// TIA Portal V19 export
DATA_BLOCK "PrjConfig_A04"   // DB212
// stored: MemoryReserve 100
   VAR
      Area04_Main : "AreaConfig";
   END_VAR
   VAR RETAIN
      A0303 : Struct
         Spalla : Struct
            Testa : Struct
               Ax : "Positioning_DOL_Machine_Config";
               DelayMissingCondition { ExternalAccessible := 'False'; ExternalVisible := 'False'; ExternalWritable := 'False'} : Time := T#0MS;
            END_STRUCT;
            Coda : Struct
               Ax : "Positioning_DOL_Machine_Config";
               DelayMissingCondition { ExternalAccessible := 'False'; ExternalVisible := 'False'; ExternalWritable := 'False'} : Time := T#0MS;
            END_STRUCT;
         END_STRUCT;
         Spintore : Struct
            Testa : Struct
               Vrt : "ValveMachine_Config";
               Orz { S7_SetPoint := 'True'} : "ValveMachine_Config";
            END_STRUCT;
            Coda : Struct
               Vrt : "ValveMachine_Config";
               Orz { S7_SetPoint := 'True'} : "ValveMachine_Config";
            END_STRUCT;
            DelayMissingCondition { ExternalAccessible := 'False'; ExternalVisible := 'False'; ExternalWritable := 'False'} : Time := T#0MS;
         END_STRUCT;
         TraslazioneStrato : Struct
            Testa : Struct
               Ax { S7_SetPoint := 'True'} : "Positioning_EPOS_Machine_Config_NEW";
               Manip_Sostegno { S7_SetPoint := 'True'} : "ValveMachine_Config";
               Manip_Pareggiatore { S7_SetPoint := 'True'} : "ValveMachine_Config";
               SostegnoVrt { S7_SetPoint := 'True'} : "ValveMachine_Config";
            END_STRUCT;
            Coda : Struct
               Ax { S7_SetPoint := 'True'} : "Positioning_EPOS_Machine_Config_NEW";
               Manip_Sostegno { S7_SetPoint := 'True'} : "ValveMachine_Config";
               Manip_Pareggiatore { S7_SetPoint := 'True'} : "ValveMachine_Config";
               SostegnoVrt { S7_SetPoint := 'True'} : "ValveMachine_Config";
               DelayMissingCondition { ExternalAccessible := 'False'; ExternalVisible := 'False'; ExternalWritable := 'False'} : Time := T#0MS;
            END_STRUCT;
            DelayMissingCondition { ExternalAccessible := 'False'; ExternalVisible := 'False'; ExternalWritable := 'False'} : Time := T#2S;
         END_STRUCT;
         Sollevamento : Struct
            Testa : Struct
               Ax : "Positioning_DOL_Machine_Config";
            END_STRUCT;
            Coda : Struct
               Ax : "Positioning_DOL_Machine_Config";
            END_STRUCT;
            DelayMissingCondition { ExternalAccessible := 'False'; ExternalVisible := 'False'; ExternalWritable := 'False'} : Time := T#0MS;
         END_STRUCT;
         Sostegno : Struct
            Testa : Struct
               Ax : "Positioning_DOL_Machine_Config";
               V_1 { S7_SetPoint := 'True'} : "ValveMachine_Config";
               V_2 { S7_SetPoint := 'True'} : "ValveMachine_Config";
               DelayMissingCondition { ExternalAccessible := 'False'; ExternalVisible := 'False'; ExternalWritable := 'False'} : Time := T#0MS;
            END_STRUCT;
            Coda : Struct
               Ax : "Positioning_DOL_Machine_Config";
               V_1 { S7_SetPoint := 'True'} : "ValveMachine_Config";
               V_2 { S7_SetPoint := 'True'} : "ValveMachine_Config";
               DelayMissingCondition { ExternalAccessible := 'False'; ExternalVisible := 'False'; ExternalWritable := 'False'} : Time := T#0MS;
            END_STRUCT;
         END_STRUCT;
      END_STRUCT;
      A0304 : Struct
         Navetta : Struct
            Testa : Struct
               Ax : "Positioning_DOL_Machine_Config";
               PalettiEsterni { S7_SetPoint := 'True'} : "ValveMachine_Config";
               PalettiInterni { S7_SetPoint := 'True'} : "ValveMachine_Config";
            END_STRUCT;
            Coda : Struct
               Ax : "Positioning_DOL_Machine_Config";
               PalettiEsterni { S7_SetPoint := 'True'} : "ValveMachine_Config";
               PalettiInterni { S7_SetPoint := 'True'} : "ValveMachine_Config";
            END_STRUCT;
            DelayMissingCondition { ExternalAccessible := 'False'; ExternalVisible := 'False'; ExternalWritable := 'False'} : Time := T#0MS;
         END_STRUCT;
      END_STRUCT;
   END_VAR
BEGIN
   Area04_Main.TimeOutStopImmediate := T#1S_500MS;
   Area04_Main.TimeOutStopInPhase := T#10S;
   Area04_Main.TimeOutStopProgrammed := T#5M;
   Area04_Main.TimeOutResetAlarms := T#1S;
   A0303.Spalla.Testa.Ax.DelayMissingCondition := T#3S;
   A0303.Spalla.Testa.Ax.CyclicOBTime_ms := 10.0;
   A0303.Spalla.Testa.Ax.Ax.limitMinus := 83.0;
   A0303.Spalla.Testa.Ax.Ax.limitPlus := 2455.0;
   A0303.Spalla.Testa.Ax.Ax.Backlash := 0.0;
   A0303.Spalla.Testa.Ax.Ax.BacklashActivation := FALSE;
   A0303.Spalla.Testa.Ax.Ax.ToleranceWindow := 0.1;
   A0303.Spalla.Testa.Ax.Ax.ToleranceWindowDelay := T#100MS;
   A0303.Spalla.Testa.Ax.Ax.PreCutOff := 0.0;
   A0303.Spalla.Testa.Ax.Ax.PreEndLowSpeed := 0.0;
   A0303.Spalla.Testa.Ax.Ax.PreEndMedSpeed := 0.0;
   A0303.Spalla.Testa.Ax.Ax.ChangeDirectionDelay := T#0MS;
   A0303.Spalla.Testa.Ax.Ax.StandstillVelocity := 0.5;
   A0303.Spalla.Testa.Ax.Ax.StandStillDelay := T#100MS;
   A0303.Spalla.Testa.Ax.Ax.HomingDirection := FALSE;
   A0303.Spalla.Testa.Ax.Ax.RecallTime := 0.0;
   A0303.Spalla.Testa.Ax.Ax.VelocityFilter_T := 10.0;
   A0303.Spalla.Testa.Ax.Ax.VelocityMeasUnit := 2;
   A0303.Spalla.Testa.Ax.Ax.PosFbkDisabled := FALSE;
   A0303.Spalla.Testa.Ax.Ax.FbkCtrlDisabled := TRUE;
   A0303.Spalla.Testa.Ax.Ax_UM2."m" := 1.0;
   A0303.Spalla.Testa.Ax.Ax_UM2.q := -286.0;
   A0303.Spalla.Testa.Ax.S120.SpeedMotor.ReferenceVelocity := 2000.0;
   A0303.Spalla.Testa.Ax.S120.SpeedMotor.InvertDirection := FALSE;
   A0303.Spalla.Testa.Ax.S120.PowerOffDelay := T#5S;
   A0303.Spalla.Testa.Ax.S120.StandstillVelocity := 50.0;
   A0303.Spalla.Testa.Ax.S120.AccTime := 0.25;
   A0303.Spalla.Testa.Ax.S120.DecTime := 0.25;
   A0303.Spalla.Testa.Ax.Fan.Presence := FALSE;
   A0303.Spalla.Testa.Ax.Fan.DelayOff := T#10M;
   A0303.Spalla.Testa.Ax.Brake_Presence := FALSE;
   A0303.Spalla.Coda.Ax.DelayMissingCondition := T#3S;
   A0303.Spalla.Coda.Ax.CyclicOBTime_ms := 10.0;
   A0303.Spalla.Coda.Ax.Ax.limitMinus := 80.0;
   A0303.Spalla.Coda.Ax.Ax.limitPlus := 2455.0;
   A0303.Spalla.Coda.Ax.Ax.Backlash := 0.0;
   A0303.Spalla.Coda.Ax.Ax.BacklashActivation := FALSE;
   A0303.Spalla.Coda.Ax.Ax.ToleranceWindow := 0.1;
   A0303.Spalla.Coda.Ax.Ax.ToleranceWindowDelay := T#100MS;
   A0303.Spalla.Coda.Ax.Ax.PreCutOff := 0.0;
   A0303.Spalla.Coda.Ax.Ax.PreEndLowSpeed := 0.0;
   A0303.Spalla.Coda.Ax.Ax.PreEndMedSpeed := 0.0;
   A0303.Spalla.Coda.Ax.Ax.ChangeDirectionDelay := T#0MS;
   A0303.Spalla.Coda.Ax.Ax.StandstillVelocity := 0.5;
   A0303.Spalla.Coda.Ax.Ax.StandStillDelay := T#100MS;
   A0303.Spalla.Coda.Ax.Ax.HomingDirection := FALSE;
   A0303.Spalla.Coda.Ax.Ax.RecallTime := 0.0;
   A0303.Spalla.Coda.Ax.Ax.VelocityFilter_T := 10.0;
   A0303.Spalla.Coda.Ax.Ax.VelocityMeasUnit := 2;
   A0303.Spalla.Coda.Ax.Ax.PosFbkDisabled := FALSE;
   A0303.Spalla.Coda.Ax.Ax.FbkCtrlDisabled := TRUE;
   A0303.Spalla.Coda.Ax.Ax_UM2."m" := 1.0;
   A0303.Spalla.Coda.Ax.Ax_UM2.q := -286.0;
   A0303.Spalla.Coda.Ax.S120.SpeedMotor.ReferenceVelocity := 2000.0;
   A0303.Spalla.Coda.Ax.S120.SpeedMotor.InvertDirection := FALSE;
   A0303.Spalla.Coda.Ax.S120.PowerOffDelay := T#5S;
   A0303.Spalla.Coda.Ax.S120.StandstillVelocity := 50.0;
   A0303.Spalla.Coda.Ax.S120.AccTime := 0.25;
   A0303.Spalla.Coda.Ax.S120.DecTime := 0.25;
   A0303.Spalla.Coda.Ax.Fan.Presence := FALSE;
   A0303.Spalla.Coda.Ax.Fan.DelayOff := T#10M;
   A0303.Spalla.Coda.Ax.Brake_Presence := FALSE;
   A0303.Spintore.Testa.Vrt.DelayPressureRunningTimeout := T#3S;
   A0303.Spintore.Testa.Vrt.DelayMissingCondition := T#3S;
   A0303.Spintore.Testa.Vrt.Rest_LsQty := 1;
   A0303.Spintore.Testa.Vrt.Work_LsQty := 1;
   A0303.Spintore.Testa.Vrt.Rest_RetainAut := FALSE;
   A0303.Spintore.Testa.Vrt.Work_RetainAut := FALSE;
   A0303.Spintore.Testa.Vrt.V.RestLimSwitchExist := TRUE;
   A0303.Spintore.Testa.Vrt.V.WorkLimSwitchExist := TRUE;
   A0303.Spintore.Testa.Vrt.V.CheckOilInPressure := FALSE;
   A0303.Spintore.Testa.Vrt.V.CutRestWhenIsAtRest := TRUE;
   A0303.Spintore.Testa.Vrt.V.CutWorkWhenIsAtWork := TRUE;
   A0303.Spintore.Testa.Vrt.V.RestTime := T#0MS;
   A0303.Spintore.Testa.Vrt.V.WorkTime := T#0MS;
   A0303.Spintore.Testa.Vrt.V.RestTimeOut := T#2S;
   A0303.Spintore.Testa.Vrt.V.WorkTimeOut := T#2S;
   A0303.Spintore.Testa.Orz.DelayPressureRunningTimeout := T#3S;
   A0303.Spintore.Testa.Orz.DelayMissingCondition := T#3S;
   A0303.Spintore.Testa.Orz.Rest_LsQty := 1;
   A0303.Spintore.Testa.Orz.Work_LsQty := 1;
   A0303.Spintore.Testa.Orz.Rest_RetainAut := FALSE;
   A0303.Spintore.Testa.Orz.Work_RetainAut := FALSE;
   A0303.Spintore.Testa.Orz.V.RestLimSwitchExist := TRUE;
   A0303.Spintore.Testa.Orz.V.WorkLimSwitchExist := TRUE;
   A0303.Spintore.Testa.Orz.V.CheckOilInPressure := FALSE;
   A0303.Spintore.Testa.Orz.V.CutRestWhenIsAtRest := TRUE;
   A0303.Spintore.Testa.Orz.V.CutWorkWhenIsAtWork := TRUE;
   A0303.Spintore.Testa.Orz.V.RestTime := T#0MS;
   A0303.Spintore.Testa.Orz.V.WorkTime := T#0MS;
   A0303.Spintore.Testa.Orz.V.RestTimeOut := T#2S;
   A0303.Spintore.Testa.Orz.V.WorkTimeOut := T#2S;
   A0303.Spintore.Coda.Vrt.DelayPressureRunningTimeout := T#3S;
   A0303.Spintore.Coda.Vrt.DelayMissingCondition := T#3S;
   A0303.Spintore.Coda.Vrt.Rest_LsQty := 1;
   A0303.Spintore.Coda.Vrt.Work_LsQty := 1;
   A0303.Spintore.Coda.Vrt.Rest_RetainAut := FALSE;
   A0303.Spintore.Coda.Vrt.Work_RetainAut := FALSE;
   A0303.Spintore.Coda.Vrt.V.RestLimSwitchExist := TRUE;
   A0303.Spintore.Coda.Vrt.V.WorkLimSwitchExist := TRUE;
   A0303.Spintore.Coda.Vrt.V.CheckOilInPressure := FALSE;
   A0303.Spintore.Coda.Vrt.V.CutRestWhenIsAtRest := TRUE;
   A0303.Spintore.Coda.Vrt.V.CutWorkWhenIsAtWork := TRUE;
   A0303.Spintore.Coda.Vrt.V.RestTime := T#0MS;
   A0303.Spintore.Coda.Vrt.V.WorkTime := T#0MS;
   A0303.Spintore.Coda.Vrt.V.RestTimeOut := T#2S;
   A0303.Spintore.Coda.Vrt.V.WorkTimeOut := T#2S;
   A0303.Spintore.Coda.Orz.DelayPressureRunningTimeout := T#3S;
   A0303.Spintore.Coda.Orz.DelayMissingCondition := T#3S;
   A0303.Spintore.Coda.Orz.Rest_LsQty := 1;
   A0303.Spintore.Coda.Orz.Work_LsQty := 1;
   A0303.Spintore.Coda.Orz.Rest_RetainAut := FALSE;
   A0303.Spintore.Coda.Orz.Work_RetainAut := FALSE;
   A0303.Spintore.Coda.Orz.V.RestLimSwitchExist := TRUE;
   A0303.Spintore.Coda.Orz.V.WorkLimSwitchExist := TRUE;
   A0303.Spintore.Coda.Orz.V.CheckOilInPressure := FALSE;
   A0303.Spintore.Coda.Orz.V.CutRestWhenIsAtRest := TRUE;
   A0303.Spintore.Coda.Orz.V.CutWorkWhenIsAtWork := TRUE;
   A0303.Spintore.Coda.Orz.V.RestTime := T#0MS;
   A0303.Spintore.Coda.Orz.V.WorkTime := T#0MS;
   A0303.Spintore.Coda.Orz.V.RestTimeOut := T#2S;
   A0303.Spintore.Coda.Orz.V.WorkTimeOut := T#2S;
   A0303.TraslazioneStrato.Testa.Ax.SLS_Vel := 0.0;
   A0303.TraslazioneStrato.Testa.Ax.DelayMissingCondition := T#2S;
   A0303.TraslazioneStrato.Testa.Ax.Ax.Encoder_Inc_AutoReloadPosition := FALSE;
   A0303.TraslazioneStrato.Testa.Ax.Ax.Encoder_is_Absolute := TRUE;
   A0303.TraslazioneStrato.Testa.Ax.Ax.LeadScrewPitchVal := 9.9996894;
   A0303.TraslazioneStrato.Testa.Ax.Ax.MotorRevolution := 20.0;
   A0303.TraslazioneStrato.Testa.Ax.Ax.LoadRevolution := 1.0;
   A0303.TraslazioneStrato.Testa.Ax.Ax.PowerOffDelay := T#2S;
   A0303.TraslazioneStrato.Testa.Ax.Ax.MaxRPM_S120_P2000 := 6000.0;
   A0303.TraslazioneStrato.Testa.Ax.Ax.MaxVel_S120_P2571 := 60000.0;
   A0303.TraslazioneStrato.Testa.Ax.Ax.MaxAcc_S120_P2572 := 4000.0;
   A0303.TraslazioneStrato.Testa.Ax.Ax.MaxDec_S120_P2573 := 4000.0;
   A0303.TraslazioneStrato.Testa.Ax.Ax.Modulo_S120_P2566 := 0.0;
   A0303.TraslazioneStrato.Testa.Ax.Ax.SwLimMinus_S120_P2580 := -1015.0;
   A0303.TraslazioneStrato.Testa.Ax.Ax.SwLimPlus_S120_P2581 := 10.0;
   A0303.TraslazioneStrato.Testa.Ax.Fan.Presence := FALSE;
   A0303.TraslazioneStrato.Testa.Ax.Fan.DelayOff := T#0MS;
   A0303.TraslazioneStrato.Testa.Ax.Brake_Presence := FALSE;
   A0303.TraslazioneStrato.Testa.Manip_Sostegno.DelayPressureRunningTimeout := T#3S;
   A0303.TraslazioneStrato.Testa.Manip_Sostegno.DelayMissingCondition := T#3S;
   A0303.TraslazioneStrato.Testa.Manip_Sostegno.Rest_LsQty := 1;
   A0303.TraslazioneStrato.Testa.Manip_Sostegno.Work_LsQty := 1;
   A0303.TraslazioneStrato.Testa.Manip_Sostegno.Rest_RetainAut := FALSE;
   A0303.TraslazioneStrato.Testa.Manip_Sostegno.Work_RetainAut := FALSE;
   A0303.TraslazioneStrato.Testa.Manip_Sostegno.V.RestLimSwitchExist := TRUE;
   A0303.TraslazioneStrato.Testa.Manip_Sostegno.V.WorkLimSwitchExist := TRUE;
   A0303.TraslazioneStrato.Testa.Manip_Sostegno.V.CheckOilInPressure := FALSE;
   A0303.TraslazioneStrato.Testa.Manip_Sostegno.V.CutRestWhenIsAtRest := TRUE;
   A0303.TraslazioneStrato.Testa.Manip_Sostegno.V.CutWorkWhenIsAtWork := TRUE;
   A0303.TraslazioneStrato.Testa.Manip_Sostegno.V.RestTime := T#0MS;
   A0303.TraslazioneStrato.Testa.Manip_Sostegno.V.WorkTime := T#0MS;
   A0303.TraslazioneStrato.Testa.Manip_Sostegno.V.RestTimeOut := T#2S;
   A0303.TraslazioneStrato.Testa.Manip_Sostegno.V.WorkTimeOut := T#2S;
   A0303.TraslazioneStrato.Testa.Manip_Pareggiatore.DelayPressureRunningTimeout := T#3S;
   A0303.TraslazioneStrato.Testa.Manip_Pareggiatore.DelayMissingCondition := T#3S;
   A0303.TraslazioneStrato.Testa.Manip_Pareggiatore.Rest_LsQty := 1;
   A0303.TraslazioneStrato.Testa.Manip_Pareggiatore.Work_LsQty := 1;
   A0303.TraslazioneStrato.Testa.Manip_Pareggiatore.Rest_RetainAut := FALSE;
   A0303.TraslazioneStrato.Testa.Manip_Pareggiatore.Work_RetainAut := FALSE;
   A0303.TraslazioneStrato.Testa.Manip_Pareggiatore.V.RestLimSwitchExist := TRUE;
   A0303.TraslazioneStrato.Testa.Manip_Pareggiatore.V.WorkLimSwitchExist := TRUE;
   A0303.TraslazioneStrato.Testa.Manip_Pareggiatore.V.CheckOilInPressure := FALSE;
   A0303.TraslazioneStrato.Testa.Manip_Pareggiatore.V.CutRestWhenIsAtRest := TRUE;
   A0303.TraslazioneStrato.Testa.Manip_Pareggiatore.V.CutWorkWhenIsAtWork := TRUE;
   A0303.TraslazioneStrato.Testa.Manip_Pareggiatore.V.RestTime := T#0MS;
   A0303.TraslazioneStrato.Testa.Manip_Pareggiatore.V.WorkTime := T#0MS;
   A0303.TraslazioneStrato.Testa.Manip_Pareggiatore.V.RestTimeOut := T#2S;
   A0303.TraslazioneStrato.Testa.Manip_Pareggiatore.V.WorkTimeOut := T#2S;
   A0303.TraslazioneStrato.Testa.SostegnoVrt.DelayPressureRunningTimeout := T#3S;
   A0303.TraslazioneStrato.Testa.SostegnoVrt.DelayMissingCondition := T#3S;
   A0303.TraslazioneStrato.Testa.SostegnoVrt.Rest_LsQty := 0;
   A0303.TraslazioneStrato.Testa.SostegnoVrt.Work_LsQty := 0;
   A0303.TraslazioneStrato.Testa.SostegnoVrt.Rest_RetainAut := FALSE;
   A0303.TraslazioneStrato.Testa.SostegnoVrt.Work_RetainAut := FALSE;
   A0303.TraslazioneStrato.Testa.SostegnoVrt.V.RestLimSwitchExist := TRUE;
   A0303.TraslazioneStrato.Testa.SostegnoVrt.V.WorkLimSwitchExist := TRUE;
   A0303.TraslazioneStrato.Testa.SostegnoVrt.V.CheckOilInPressure := FALSE;
   A0303.TraslazioneStrato.Testa.SostegnoVrt.V.CutRestWhenIsAtRest := TRUE;
   A0303.TraslazioneStrato.Testa.SostegnoVrt.V.CutWorkWhenIsAtWork := TRUE;
   A0303.TraslazioneStrato.Testa.SostegnoVrt.V.RestTime := T#0MS;
   A0303.TraslazioneStrato.Testa.SostegnoVrt.V.WorkTime := T#0MS;
   A0303.TraslazioneStrato.Testa.SostegnoVrt.V.RestTimeOut := T#1H;
   A0303.TraslazioneStrato.Testa.SostegnoVrt.V.WorkTimeOut := T#1H;
   A0303.TraslazioneStrato.Coda.Ax.SLS_Vel := 0.0;
   A0303.TraslazioneStrato.Coda.Ax.DelayMissingCondition := T#2S;
   A0303.TraslazioneStrato.Coda.Ax.Ax.Encoder_Inc_AutoReloadPosition := FALSE;
   A0303.TraslazioneStrato.Coda.Ax.Ax.Encoder_is_Absolute := TRUE;
   A0303.TraslazioneStrato.Coda.Ax.Ax.LeadScrewPitchVal := 9.9996894;
   A0303.TraslazioneStrato.Coda.Ax.Ax.MotorRevolution := 20.0;
   A0303.TraslazioneStrato.Coda.Ax.Ax.LoadRevolution := 1.0;
   A0303.TraslazioneStrato.Coda.Ax.Ax.PowerOffDelay := T#2S;
   A0303.TraslazioneStrato.Coda.Ax.Ax.MaxRPM_S120_P2000 := 6000.0;
   A0303.TraslazioneStrato.Coda.Ax.Ax.MaxVel_S120_P2571 := 60000.0;
   A0303.TraslazioneStrato.Coda.Ax.Ax.MaxAcc_S120_P2572 := 4000.0;
   A0303.TraslazioneStrato.Coda.Ax.Ax.MaxDec_S120_P2573 := 4000.0;
   A0303.TraslazioneStrato.Coda.Ax.Ax.Modulo_S120_P2566 := 0.0;
   A0303.TraslazioneStrato.Coda.Ax.Ax.SwLimMinus_S120_P2580 := -1015.0;
   A0303.TraslazioneStrato.Coda.Ax.Ax.SwLimPlus_S120_P2581 := 10.0;
   A0303.TraslazioneStrato.Coda.Ax.Fan.Presence := FALSE;
   A0303.TraslazioneStrato.Coda.Ax.Fan.DelayOff := T#0MS;
   A0303.TraslazioneStrato.Coda.Ax.Brake_Presence := FALSE;
   A0303.TraslazioneStrato.Coda.Manip_Sostegno.DelayPressureRunningTimeout := T#3S;
   A0303.TraslazioneStrato.Coda.Manip_Sostegno.DelayMissingCondition := T#3S;
   A0303.TraslazioneStrato.Coda.Manip_Sostegno.Rest_LsQty := 1;
   A0303.TraslazioneStrato.Coda.Manip_Sostegno.Work_LsQty := 1;
   A0303.TraslazioneStrato.Coda.Manip_Sostegno.Rest_RetainAut := FALSE;
   A0303.TraslazioneStrato.Coda.Manip_Sostegno.Work_RetainAut := FALSE;
   A0303.TraslazioneStrato.Coda.Manip_Sostegno.V.RestLimSwitchExist := TRUE;
   A0303.TraslazioneStrato.Coda.Manip_Sostegno.V.WorkLimSwitchExist := TRUE;
   A0303.TraslazioneStrato.Coda.Manip_Sostegno.V.CheckOilInPressure := FALSE;
   A0303.TraslazioneStrato.Coda.Manip_Sostegno.V.CutRestWhenIsAtRest := TRUE;
   A0303.TraslazioneStrato.Coda.Manip_Sostegno.V.CutWorkWhenIsAtWork := TRUE;
   A0303.TraslazioneStrato.Coda.Manip_Sostegno.V.RestTime := T#0MS;
   A0303.TraslazioneStrato.Coda.Manip_Sostegno.V.WorkTime := T#0MS;
   A0303.TraslazioneStrato.Coda.Manip_Sostegno.V.RestTimeOut := T#2S;
   A0303.TraslazioneStrato.Coda.Manip_Sostegno.V.WorkTimeOut := T#2S;
   A0303.TraslazioneStrato.Coda.Manip_Pareggiatore.DelayPressureRunningTimeout := T#3S;
   A0303.TraslazioneStrato.Coda.Manip_Pareggiatore.DelayMissingCondition := T#3S;
   A0303.TraslazioneStrato.Coda.Manip_Pareggiatore.Rest_LsQty := 1;
   A0303.TraslazioneStrato.Coda.Manip_Pareggiatore.Work_LsQty := 1;
   A0303.TraslazioneStrato.Coda.Manip_Pareggiatore.Rest_RetainAut := FALSE;
   A0303.TraslazioneStrato.Coda.Manip_Pareggiatore.Work_RetainAut := FALSE;
   A0303.TraslazioneStrato.Coda.Manip_Pareggiatore.V.RestLimSwitchExist := TRUE;
   A0303.TraslazioneStrato.Coda.Manip_Pareggiatore.V.WorkLimSwitchExist := TRUE;
   A0303.TraslazioneStrato.Coda.Manip_Pareggiatore.V.CheckOilInPressure := FALSE;
   A0303.TraslazioneStrato.Coda.Manip_Pareggiatore.V.CutRestWhenIsAtRest := TRUE;
   A0303.TraslazioneStrato.Coda.Manip_Pareggiatore.V.CutWorkWhenIsAtWork := TRUE;
   A0303.TraslazioneStrato.Coda.Manip_Pareggiatore.V.RestTime := T#0MS;
   A0303.TraslazioneStrato.Coda.Manip_Pareggiatore.V.WorkTime := T#0MS;
   A0303.TraslazioneStrato.Coda.Manip_Pareggiatore.V.RestTimeOut := T#2S;
   A0303.TraslazioneStrato.Coda.Manip_Pareggiatore.V.WorkTimeOut := T#2S;
   A0303.TraslazioneStrato.Coda.SostegnoVrt.DelayPressureRunningTimeout := T#3S;
   A0303.TraslazioneStrato.Coda.SostegnoVrt.DelayMissingCondition := T#3S;
   A0303.TraslazioneStrato.Coda.SostegnoVrt.Rest_LsQty := 0;
   A0303.TraslazioneStrato.Coda.SostegnoVrt.Work_LsQty := 0;
   A0303.TraslazioneStrato.Coda.SostegnoVrt.Rest_RetainAut := FALSE;
   A0303.TraslazioneStrato.Coda.SostegnoVrt.Work_RetainAut := FALSE;
   A0303.TraslazioneStrato.Coda.SostegnoVrt.V.RestLimSwitchExist := TRUE;
   A0303.TraslazioneStrato.Coda.SostegnoVrt.V.WorkLimSwitchExist := TRUE;
   A0303.TraslazioneStrato.Coda.SostegnoVrt.V.CheckOilInPressure := FALSE;
   A0303.TraslazioneStrato.Coda.SostegnoVrt.V.CutRestWhenIsAtRest := TRUE;
   A0303.TraslazioneStrato.Coda.SostegnoVrt.V.CutWorkWhenIsAtWork := TRUE;
   A0303.TraslazioneStrato.Coda.SostegnoVrt.V.RestTime := T#0MS;
   A0303.TraslazioneStrato.Coda.SostegnoVrt.V.WorkTime := T#0MS;
   A0303.TraslazioneStrato.Coda.SostegnoVrt.V.RestTimeOut := T#1H;
   A0303.TraslazioneStrato.Coda.SostegnoVrt.V.WorkTimeOut := T#1H;
   A0303.Sollevamento.Testa.Ax.DelayMissingCondition := T#3S;
   A0303.Sollevamento.Testa.Ax.CyclicOBTime_ms := 10.0;
   A0303.Sollevamento.Testa.Ax.Ax.limitMinus := 0.0;
   A0303.Sollevamento.Testa.Ax.Ax.limitPlus := 476.0;
   A0303.Sollevamento.Testa.Ax.Ax.Backlash := 0.0;
   A0303.Sollevamento.Testa.Ax.Ax.BacklashActivation := FALSE;
   A0303.Sollevamento.Testa.Ax.Ax.ToleranceWindow := 0.1;
   A0303.Sollevamento.Testa.Ax.Ax.ToleranceWindowDelay := T#100MS;
   A0303.Sollevamento.Testa.Ax.Ax.PreCutOff := 0.0;
   A0303.Sollevamento.Testa.Ax.Ax.PreEndLowSpeed := 0.0;
   A0303.Sollevamento.Testa.Ax.Ax.PreEndMedSpeed := 0.0;
   A0303.Sollevamento.Testa.Ax.Ax.ChangeDirectionDelay := T#0MS;
   A0303.Sollevamento.Testa.Ax.Ax.StandstillVelocity := 0.5;
   A0303.Sollevamento.Testa.Ax.Ax.StandStillDelay := T#100MS;
   A0303.Sollevamento.Testa.Ax.Ax.HomingDirection := FALSE;
   A0303.Sollevamento.Testa.Ax.Ax.RecallTime := 0.0;
   A0303.Sollevamento.Testa.Ax.Ax.VelocityFilter_T := 10.0;
   A0303.Sollevamento.Testa.Ax.Ax.VelocityMeasUnit := 2;
   A0303.Sollevamento.Testa.Ax.Ax.PosFbkDisabled := FALSE;
   A0303.Sollevamento.Testa.Ax.Ax.FbkCtrlDisabled := TRUE;
   A0303.Sollevamento.Testa.Ax.Ax_UM2."m" := 1.0;
   A0303.Sollevamento.Testa.Ax.Ax_UM2.q := 0.0;
   A0303.Sollevamento.Testa.Ax.S120.SpeedMotor.ReferenceVelocity := 2000.0;
   A0303.Sollevamento.Testa.Ax.S120.SpeedMotor.InvertDirection := FALSE;
   A0303.Sollevamento.Testa.Ax.S120.PowerOffDelay := T#5S;
   A0303.Sollevamento.Testa.Ax.S120.StandstillVelocity := 50.0;
   A0303.Sollevamento.Testa.Ax.S120.AccTime := 0.25;
   A0303.Sollevamento.Testa.Ax.S120.DecTime := 0.25;
   A0303.Sollevamento.Testa.Ax.Fan.Presence := FALSE;
   A0303.Sollevamento.Testa.Ax.Fan.DelayOff := T#10M;
   A0303.Sollevamento.Testa.Ax.Brake_Presence := FALSE;
   A0303.Sollevamento.Coda.Ax.DelayMissingCondition := T#3S;
   A0303.Sollevamento.Coda.Ax.CyclicOBTime_ms := 10.0;
   A0303.Sollevamento.Coda.Ax.Ax.limitMinus := 0.0;
   A0303.Sollevamento.Coda.Ax.Ax.limitPlus := 476.0;
   A0303.Sollevamento.Coda.Ax.Ax.Backlash := 0.0;
   A0303.Sollevamento.Coda.Ax.Ax.BacklashActivation := FALSE;
   A0303.Sollevamento.Coda.Ax.Ax.ToleranceWindow := 0.1;
   A0303.Sollevamento.Coda.Ax.Ax.ToleranceWindowDelay := T#100MS;
   A0303.Sollevamento.Coda.Ax.Ax.PreCutOff := 0.0;
   A0303.Sollevamento.Coda.Ax.Ax.PreEndLowSpeed := 0.0;
   A0303.Sollevamento.Coda.Ax.Ax.PreEndMedSpeed := 0.0;
   A0303.Sollevamento.Coda.Ax.Ax.ChangeDirectionDelay := T#0MS;
   A0303.Sollevamento.Coda.Ax.Ax.StandstillVelocity := 0.5;
   A0303.Sollevamento.Coda.Ax.Ax.StandStillDelay := T#100MS;
   A0303.Sollevamento.Coda.Ax.Ax.HomingDirection := FALSE;
   A0303.Sollevamento.Coda.Ax.Ax.RecallTime := 0.0;
   A0303.Sollevamento.Coda.Ax.Ax.VelocityFilter_T := 10.0;
   A0303.Sollevamento.Coda.Ax.Ax.VelocityMeasUnit := 2;
   A0303.Sollevamento.Coda.Ax.Ax.PosFbkDisabled := FALSE;
   A0303.Sollevamento.Coda.Ax.Ax.FbkCtrlDisabled := TRUE;
   A0303.Sollevamento.Coda.Ax.Ax_UM2."m" := 1.0;
   A0303.Sollevamento.Coda.Ax.Ax_UM2.q := 0.0;
   A0303.Sollevamento.Coda.Ax.S120.SpeedMotor.ReferenceVelocity := 2000.0;
   A0303.Sollevamento.Coda.Ax.S120.SpeedMotor.InvertDirection := FALSE;
   A0303.Sollevamento.Coda.Ax.S120.PowerOffDelay := T#5S;
   A0303.Sollevamento.Coda.Ax.S120.StandstillVelocity := 50.0;
   A0303.Sollevamento.Coda.Ax.S120.AccTime := 0.25;
   A0303.Sollevamento.Coda.Ax.S120.DecTime := 0.25;
   A0303.Sollevamento.Coda.Ax.Fan.Presence := FALSE;
   A0303.Sollevamento.Coda.Ax.Fan.DelayOff := T#10M;
   A0303.Sollevamento.Coda.Ax.Brake_Presence := FALSE;
   A0303.Sostegno.Testa.Ax.DelayMissingCondition := T#3S;
   A0303.Sostegno.Testa.Ax.CyclicOBTime_ms := 10.0;
   A0303.Sostegno.Testa.Ax.Ax.limitMinus := 419.0;
   A0303.Sostegno.Testa.Ax.Ax.limitPlus := 689.0;
   A0303.Sostegno.Testa.Ax.Ax.Backlash := 0.0;
   A0303.Sostegno.Testa.Ax.Ax.BacklashActivation := FALSE;
   A0303.Sostegno.Testa.Ax.Ax.ToleranceWindow := 0.1;
   A0303.Sostegno.Testa.Ax.Ax.ToleranceWindowDelay := T#100MS;
   A0303.Sostegno.Testa.Ax.Ax.PreCutOff := 0.0;
   A0303.Sostegno.Testa.Ax.Ax.PreEndLowSpeed := 0.0;
   A0303.Sostegno.Testa.Ax.Ax.PreEndMedSpeed := 0.0;
   A0303.Sostegno.Testa.Ax.Ax.ChangeDirectionDelay := T#0MS;
   A0303.Sostegno.Testa.Ax.Ax.StandstillVelocity := 0.5;
   A0303.Sostegno.Testa.Ax.Ax.StandStillDelay := T#100MS;
   A0303.Sostegno.Testa.Ax.Ax.HomingDirection := FALSE;
   A0303.Sostegno.Testa.Ax.Ax.RecallTime := 0.0;
   A0303.Sostegno.Testa.Ax.Ax.VelocityFilter_T := 10.0;
   A0303.Sostegno.Testa.Ax.Ax.VelocityMeasUnit := 2;
   A0303.Sostegno.Testa.Ax.Ax.PosFbkDisabled := FALSE;
   A0303.Sostegno.Testa.Ax.Ax.FbkCtrlDisabled := TRUE;
   A0303.Sostegno.Testa.Ax.Ax_UM2."m" := 1.0;
   A0303.Sostegno.Testa.Ax.Ax_UM2.q := 0.0;
   A0303.Sostegno.Testa.Ax.S120.SpeedMotor.ReferenceVelocity := 2000.0;
   A0303.Sostegno.Testa.Ax.S120.SpeedMotor.InvertDirection := FALSE;
   A0303.Sostegno.Testa.Ax.S120.PowerOffDelay := T#5S;
   A0303.Sostegno.Testa.Ax.S120.StandstillVelocity := 50.0;
   A0303.Sostegno.Testa.Ax.S120.AccTime := 0.25;
   A0303.Sostegno.Testa.Ax.S120.DecTime := 0.25;
   A0303.Sostegno.Testa.Ax.Fan.Presence := FALSE;
   A0303.Sostegno.Testa.Ax.Fan.DelayOff := T#10M;
   A0303.Sostegno.Testa.Ax.Brake_Presence := FALSE;
   A0303.Sostegno.Testa.V_1.DelayPressureRunningTimeout := T#3S;
   A0303.Sostegno.Testa.V_1.DelayMissingCondition := T#3S;
   A0303.Sostegno.Testa.V_1.Rest_LsQty := 1;
   A0303.Sostegno.Testa.V_1.Work_LsQty := 1;
   A0303.Sostegno.Testa.V_1.Rest_RetainAut := FALSE;
   A0303.Sostegno.Testa.V_1.Work_RetainAut := FALSE;
   A0303.Sostegno.Testa.V_1.V.RestLimSwitchExist := FALSE;
   A0303.Sostegno.Testa.V_1.V.WorkLimSwitchExist := FALSE;
   A0303.Sostegno.Testa.V_1.V.CheckOilInPressure := FALSE;
   A0303.Sostegno.Testa.V_1.V.CutRestWhenIsAtRest := FALSE;
   A0303.Sostegno.Testa.V_1.V.CutWorkWhenIsAtWork := FALSE;
   A0303.Sostegno.Testa.V_1.V.RestTime := T#20S;
   A0303.Sostegno.Testa.V_1.V.WorkTime := T#20S;
   A0303.Sostegno.Testa.V_1.V.RestTimeOut := T#10S;
   A0303.Sostegno.Testa.V_1.V.WorkTimeOut := T#10S;
   A0303.Sostegno.Testa.V_2.DelayPressureRunningTimeout := T#3S;
   A0303.Sostegno.Testa.V_2.DelayMissingCondition := T#3S;
   A0303.Sostegno.Testa.V_2.Rest_LsQty := 1;
   A0303.Sostegno.Testa.V_2.Work_LsQty := 1;
   A0303.Sostegno.Testa.V_2.Rest_RetainAut := FALSE;
   A0303.Sostegno.Testa.V_2.Work_RetainAut := FALSE;
   A0303.Sostegno.Testa.V_2.V.RestLimSwitchExist := FALSE;
   A0303.Sostegno.Testa.V_2.V.WorkLimSwitchExist := FALSE;
   A0303.Sostegno.Testa.V_2.V.CheckOilInPressure := FALSE;
   A0303.Sostegno.Testa.V_2.V.CutRestWhenIsAtRest := FALSE;
   A0303.Sostegno.Testa.V_2.V.CutWorkWhenIsAtWork := FALSE;
   A0303.Sostegno.Testa.V_2.V.RestTime := T#20S;
   A0303.Sostegno.Testa.V_2.V.WorkTime := T#20S;
   A0303.Sostegno.Testa.V_2.V.RestTimeOut := T#20S;
   A0303.Sostegno.Testa.V_2.V.WorkTimeOut := T#20S;
   A0303.Sostegno.Coda.Ax.DelayMissingCondition := T#3S;
   A0303.Sostegno.Coda.Ax.CyclicOBTime_ms := 10.0;
   A0303.Sostegno.Coda.Ax.Ax.limitMinus := 419.0;
   A0303.Sostegno.Coda.Ax.Ax.limitPlus := 689.0;
   A0303.Sostegno.Coda.Ax.Ax.Backlash := 0.0;
   A0303.Sostegno.Coda.Ax.Ax.BacklashActivation := FALSE;
   A0303.Sostegno.Coda.Ax.Ax.ToleranceWindow := 0.1;
   A0303.Sostegno.Coda.Ax.Ax.ToleranceWindowDelay := T#100MS;
   A0303.Sostegno.Coda.Ax.Ax.PreCutOff := 0.0;
   A0303.Sostegno.Coda.Ax.Ax.PreEndLowSpeed := 0.0;
   A0303.Sostegno.Coda.Ax.Ax.PreEndMedSpeed := 0.0;
   A0303.Sostegno.Coda.Ax.Ax.ChangeDirectionDelay := T#0MS;
   A0303.Sostegno.Coda.Ax.Ax.StandstillVelocity := 0.5;
   A0303.Sostegno.Coda.Ax.Ax.StandStillDelay := T#100MS;
   A0303.Sostegno.Coda.Ax.Ax.HomingDirection := FALSE;
   A0303.Sostegno.Coda.Ax.Ax.RecallTime := 0.0;
   A0303.Sostegno.Coda.Ax.Ax.VelocityFilter_T := 10.0;
   A0303.Sostegno.Coda.Ax.Ax.VelocityMeasUnit := 2;
   A0303.Sostegno.Coda.Ax.Ax.PosFbkDisabled := FALSE;
   A0303.Sostegno.Coda.Ax.Ax.FbkCtrlDisabled := TRUE;
   A0303.Sostegno.Coda.Ax.Ax_UM2."m" := 1.0;
   A0303.Sostegno.Coda.Ax.Ax_UM2.q := 0.0;
   A0303.Sostegno.Coda.Ax.S120.SpeedMotor.ReferenceVelocity := 2000.0;
   A0303.Sostegno.Coda.Ax.S120.SpeedMotor.InvertDirection := FALSE;
   A0303.Sostegno.Coda.Ax.S120.PowerOffDelay := T#5S;
   A0303.Sostegno.Coda.Ax.S120.StandstillVelocity := 50.0;
   A0303.Sostegno.Coda.Ax.S120.AccTime := 0.25;
   A0303.Sostegno.Coda.Ax.S120.DecTime := 0.25;
   A0303.Sostegno.Coda.Ax.Fan.Presence := FALSE;
   A0303.Sostegno.Coda.Ax.Fan.DelayOff := T#10M;
   A0303.Sostegno.Coda.Ax.Brake_Presence := FALSE;
   A0303.Sostegno.Coda.V_1.DelayPressureRunningTimeout := T#3S;
   A0303.Sostegno.Coda.V_1.DelayMissingCondition := T#3S;
   A0303.Sostegno.Coda.V_1.Rest_LsQty := 0;
   A0303.Sostegno.Coda.V_1.Work_LsQty := 0;
   A0303.Sostegno.Coda.V_1.Rest_RetainAut := FALSE;
   A0303.Sostegno.Coda.V_1.Work_RetainAut := FALSE;
   A0303.Sostegno.Coda.V_1.V.RestLimSwitchExist := FALSE;
   A0303.Sostegno.Coda.V_1.V.WorkLimSwitchExist := FALSE;
   A0303.Sostegno.Coda.V_1.V.CheckOilInPressure := FALSE;
   A0303.Sostegno.Coda.V_1.V.CutRestWhenIsAtRest := FALSE;
   A0303.Sostegno.Coda.V_1.V.CutWorkWhenIsAtWork := FALSE;
   A0303.Sostegno.Coda.V_1.V.RestTime := T#20S;
   A0303.Sostegno.Coda.V_1.V.WorkTime := T#20S;
   A0303.Sostegno.Coda.V_1.V.RestTimeOut := T#1H;
   A0303.Sostegno.Coda.V_1.V.WorkTimeOut := T#1H;
   A0303.Sostegno.Coda.V_2.DelayPressureRunningTimeout := T#3S;
   A0303.Sostegno.Coda.V_2.DelayMissingCondition := T#3S;
   A0303.Sostegno.Coda.V_2.Rest_LsQty := 0;
   A0303.Sostegno.Coda.V_2.Work_LsQty := 0;
   A0303.Sostegno.Coda.V_2.Rest_RetainAut := FALSE;
   A0303.Sostegno.Coda.V_2.Work_RetainAut := FALSE;
   A0303.Sostegno.Coda.V_2.V.RestLimSwitchExist := FALSE;
   A0303.Sostegno.Coda.V_2.V.WorkLimSwitchExist := FALSE;
   A0303.Sostegno.Coda.V_2.V.CheckOilInPressure := FALSE;
   A0303.Sostegno.Coda.V_2.V.CutRestWhenIsAtRest := FALSE;
   A0303.Sostegno.Coda.V_2.V.CutWorkWhenIsAtWork := FALSE;
   A0303.Sostegno.Coda.V_2.V.RestTime := T#20S;
   A0303.Sostegno.Coda.V_2.V.WorkTime := T#20S;
   A0303.Sostegno.Coda.V_2.V.RestTimeOut := T#1H;
   A0303.Sostegno.Coda.V_2.V.WorkTimeOut := T#1H;
   A0304.Navetta.Testa.Ax.DelayMissingCondition := T#3S;
   A0304.Navetta.Testa.Ax.CyclicOBTime_ms := 10.0;
   A0304.Navetta.Testa.Ax.Ax.limitMinus := -25.0;
   A0304.Navetta.Testa.Ax.Ax.limitPlus := 2175.0;
   A0304.Navetta.Testa.Ax.Ax.Backlash := 0.0;
   A0304.Navetta.Testa.Ax.Ax.BacklashActivation := FALSE;
   A0304.Navetta.Testa.Ax.Ax.ToleranceWindow := 0.1;
   A0304.Navetta.Testa.Ax.Ax.ToleranceWindowDelay := T#100MS;
   A0304.Navetta.Testa.Ax.Ax.PreCutOff := 0.0;
   A0304.Navetta.Testa.Ax.Ax.PreEndLowSpeed := 0.0;
   A0304.Navetta.Testa.Ax.Ax.PreEndMedSpeed := 0.0;
   A0304.Navetta.Testa.Ax.Ax.ChangeDirectionDelay := T#0MS;
   A0304.Navetta.Testa.Ax.Ax.StandstillVelocity := 0.5;
   A0304.Navetta.Testa.Ax.Ax.StandStillDelay := T#100MS;
   A0304.Navetta.Testa.Ax.Ax.HomingDirection := FALSE;
   A0304.Navetta.Testa.Ax.Ax.RecallTime := 0.0;
   A0304.Navetta.Testa.Ax.Ax.VelocityFilter_T := 10.0;
   A0304.Navetta.Testa.Ax.Ax.VelocityMeasUnit := 2;
   A0304.Navetta.Testa.Ax.Ax.PosFbkDisabled := FALSE;
   A0304.Navetta.Testa.Ax.Ax.FbkCtrlDisabled := TRUE;
   A0304.Navetta.Testa.Ax.Ax_UM2."m" := 1.0;
   A0304.Navetta.Testa.Ax.Ax_UM2.q := 0.0;
   A0304.Navetta.Testa.Ax.S120.SpeedMotor.ReferenceVelocity := 2200.0;
   A0304.Navetta.Testa.Ax.S120.SpeedMotor.InvertDirection := FALSE;
   A0304.Navetta.Testa.Ax.S120.PowerOffDelay := T#10S;
   A0304.Navetta.Testa.Ax.S120.StandstillVelocity := 20.0;
   A0304.Navetta.Testa.Ax.S120.AccTime := 2.5;
   A0304.Navetta.Testa.Ax.S120.DecTime := 2.5;
   A0304.Navetta.Testa.Ax.Fan.Presence := FALSE;
   A0304.Navetta.Testa.Ax.Fan.DelayOff := T#10M;
   A0304.Navetta.Testa.Ax.Brake_Presence := FALSE;
   A0304.Navetta.Testa.PalettiEsterni.DelayPressureRunningTimeout := T#3S;
   A0304.Navetta.Testa.PalettiEsterni.DelayMissingCondition := T#3S;
   A0304.Navetta.Testa.PalettiEsterni.Rest_LsQty := 1;
   A0304.Navetta.Testa.PalettiEsterni.Work_LsQty := 1;
   A0304.Navetta.Testa.PalettiEsterni.Rest_RetainAut := FALSE;
   A0304.Navetta.Testa.PalettiEsterni.Work_RetainAut := FALSE;
   A0304.Navetta.Testa.PalettiEsterni.V.RestLimSwitchExist := TRUE;
   A0304.Navetta.Testa.PalettiEsterni.V.WorkLimSwitchExist := FALSE;
   A0304.Navetta.Testa.PalettiEsterni.V.CheckOilInPressure := FALSE;
   A0304.Navetta.Testa.PalettiEsterni.V.CutRestWhenIsAtRest := TRUE;
   A0304.Navetta.Testa.PalettiEsterni.V.CutWorkWhenIsAtWork := TRUE;
   A0304.Navetta.Testa.PalettiEsterni.V.RestTime := T#0MS;
   A0304.Navetta.Testa.PalettiEsterni.V.WorkTime := T#500MS;
   A0304.Navetta.Testa.PalettiEsterni.V.RestTimeOut := T#6S;
   A0304.Navetta.Testa.PalettiEsterni.V.WorkTimeOut := T#6S;
   A0304.Navetta.Testa.PalettiInterni.DelayPressureRunningTimeout := T#3S;
   A0304.Navetta.Testa.PalettiInterni.DelayMissingCondition := T#3S;
   A0304.Navetta.Testa.PalettiInterni.Rest_LsQty := 1;
   A0304.Navetta.Testa.PalettiInterni.Work_LsQty := 1;
   A0304.Navetta.Testa.PalettiInterni.Rest_RetainAut := FALSE;
   A0304.Navetta.Testa.PalettiInterni.Work_RetainAut := FALSE;
   A0304.Navetta.Testa.PalettiInterni.V.RestLimSwitchExist := TRUE;
   A0304.Navetta.Testa.PalettiInterni.V.WorkLimSwitchExist := TRUE;
   A0304.Navetta.Testa.PalettiInterni.V.CheckOilInPressure := FALSE;
   A0304.Navetta.Testa.PalettiInterni.V.CutRestWhenIsAtRest := TRUE;
   A0304.Navetta.Testa.PalettiInterni.V.CutWorkWhenIsAtWork := TRUE;
   A0304.Navetta.Testa.PalettiInterni.V.RestTime := T#0MS;
   A0304.Navetta.Testa.PalettiInterni.V.WorkTime := T#0MS;
   A0304.Navetta.Testa.PalettiInterni.V.RestTimeOut := T#6S;
   A0304.Navetta.Testa.PalettiInterni.V.WorkTimeOut := T#6S;
   A0304.Navetta.Coda.Ax.DelayMissingCondition := T#3S;
   A0304.Navetta.Coda.Ax.CyclicOBTime_ms := 10.0;
   A0304.Navetta.Coda.Ax.Ax.limitMinus := -25.0;
   A0304.Navetta.Coda.Ax.Ax.limitPlus := 2175.0;
   A0304.Navetta.Coda.Ax.Ax.Backlash := 0.0;
   A0304.Navetta.Coda.Ax.Ax.BacklashActivation := FALSE;
   A0304.Navetta.Coda.Ax.Ax.ToleranceWindow := 0.1;
   A0304.Navetta.Coda.Ax.Ax.ToleranceWindowDelay := T#100MS;
   A0304.Navetta.Coda.Ax.Ax.PreCutOff := 0.0;
   A0304.Navetta.Coda.Ax.Ax.PreEndLowSpeed := 0.0;
   A0304.Navetta.Coda.Ax.Ax.PreEndMedSpeed := 0.0;
   A0304.Navetta.Coda.Ax.Ax.ChangeDirectionDelay := T#0MS;
   A0304.Navetta.Coda.Ax.Ax.StandstillVelocity := 0.5;
   A0304.Navetta.Coda.Ax.Ax.StandStillDelay := T#100MS;
   A0304.Navetta.Coda.Ax.Ax.HomingDirection := FALSE;
   A0304.Navetta.Coda.Ax.Ax.RecallTime := 0.0;
   A0304.Navetta.Coda.Ax.Ax.VelocityFilter_T := 10.0;
   A0304.Navetta.Coda.Ax.Ax.VelocityMeasUnit := 2;
   A0304.Navetta.Coda.Ax.Ax.PosFbkDisabled := FALSE;
   A0304.Navetta.Coda.Ax.Ax.FbkCtrlDisabled := TRUE;
   A0304.Navetta.Coda.Ax.Ax_UM2."m" := 1.0;
   A0304.Navetta.Coda.Ax.Ax_UM2.q := 0.0;
   A0304.Navetta.Coda.Ax.S120.SpeedMotor.ReferenceVelocity := 2200.0;
   A0304.Navetta.Coda.Ax.S120.SpeedMotor.InvertDirection := FALSE;
   A0304.Navetta.Coda.Ax.S120.PowerOffDelay := T#10S;
   A0304.Navetta.Coda.Ax.S120.StandstillVelocity := 20.0;
   A0304.Navetta.Coda.Ax.S120.AccTime := 2.5;
   A0304.Navetta.Coda.Ax.S120.DecTime := 2.5;
   A0304.Navetta.Coda.Ax.Fan.Presence := FALSE;
   A0304.Navetta.Coda.Ax.Fan.DelayOff := T#10M;
   A0304.Navetta.Coda.Ax.Brake_Presence := FALSE;
   A0304.Navetta.Coda.PalettiEsterni.DelayPressureRunningTimeout := T#3S;
   A0304.Navetta.Coda.PalettiEsterni.DelayMissingCondition := T#3S;
   A0304.Navetta.Coda.PalettiEsterni.Rest_LsQty := 1;
   A0304.Navetta.Coda.PalettiEsterni.Work_LsQty := 1;
   A0304.Navetta.Coda.PalettiEsterni.Rest_RetainAut := FALSE;
   A0304.Navetta.Coda.PalettiEsterni.Work_RetainAut := FALSE;
   A0304.Navetta.Coda.PalettiEsterni.V.RestLimSwitchExist := TRUE;
   A0304.Navetta.Coda.PalettiEsterni.V.WorkLimSwitchExist := FALSE;
   A0304.Navetta.Coda.PalettiEsterni.V.CheckOilInPressure := FALSE;
   A0304.Navetta.Coda.PalettiEsterni.V.CutRestWhenIsAtRest := TRUE;
   A0304.Navetta.Coda.PalettiEsterni.V.CutWorkWhenIsAtWork := TRUE;
   A0304.Navetta.Coda.PalettiEsterni.V.RestTime := T#0MS;
   A0304.Navetta.Coda.PalettiEsterni.V.WorkTime := T#500MS;
   A0304.Navetta.Coda.PalettiEsterni.V.RestTimeOut := T#6S;
   A0304.Navetta.Coda.PalettiEsterni.V.WorkTimeOut := T#6S;
   A0304.Navetta.Coda.PalettiInterni.DelayPressureRunningTimeout := T#3S;
   A0304.Navetta.Coda.PalettiInterni.DelayMissingCondition := T#3S;
   A0304.Navetta.Coda.PalettiInterni.Rest_LsQty := 1;
   A0304.Navetta.Coda.PalettiInterni.Work_LsQty := 1;
   A0304.Navetta.Coda.PalettiInterni.Rest_RetainAut := FALSE;
   A0304.Navetta.Coda.PalettiInterni.Work_RetainAut := FALSE;
   A0304.Navetta.Coda.PalettiInterni.V.RestLimSwitchExist := TRUE;
   A0304.Navetta.Coda.PalettiInterni.V.WorkLimSwitchExist := TRUE;
   A0304.Navetta.Coda.PalettiInterni.V.CheckOilInPressure := FALSE;
   A0304.Navetta.Coda.PalettiInterni.V.CutRestWhenIsAtRest := TRUE;
   A0304.Navetta.Coda.PalettiInterni.V.CutWorkWhenIsAtWork := TRUE;
   A0304.Navetta.Coda.PalettiInterni.V.RestTime := T#0MS;
   A0304.Navetta.Coda.PalettiInterni.V.WorkTime := T#0MS;
   A0304.Navetta.Coda.PalettiInterni.V.RestTimeOut := T#6S;
   A0304.Navetta.Coda.PalettiInterni.V.WorkTimeOut := T#6S;
END_DATA_BLOCK
